// Load stacker HW inputs
TYPE ST_HW_InputsClosedPalletCheck :
STRUCT	
	FingersLeft				: ARRAY[1..10] OF BOOL;
	FingersRight			: ARRAY[1..10] OF BOOL;	
	SensorTriggerStart		: BOOL;
	SensorTriggerStop		: BOOL;

END_STRUCT
END_TYPE

(* stored: Version 1.1.0.1, ProductVersion 3.1.4024.9
   DUT ST_HW_InputsClosedPalletCheck: Id {f9fcb07f-724b-40b5-a946-fbd0924dd5e9} *)
